SUBAPPLICATION AuxInput_Abscheider_UP (* Subapplication Type *)
  (* Standard: 61499-2 *)
  (* Version 1.0, 2023-02-06, franz *)
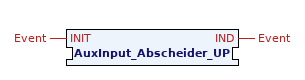
  EVENT_INPUT
    INIT;
  END_EVENT
  EVENT_OUTPUT
    IND;
  END_EVENT
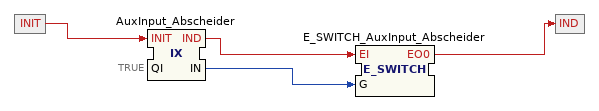
  FBS
    E_SWITCH_AuxInput_Abscheider : E_SWITCH;
    AuxInput_Abscheider : IX(QI := TRUE);
  END_FBS
  EVENT_CONNECTIONS
    AuxInput_Abscheider.IND TO E_SWITCH_AuxInput_Abscheider.EI;
    INIT TO AuxInput_Abscheider.INIT;
    E_SWITCH_AuxInput_Abscheider.EO0 TO IND;
  END_CONNECTIONS
  DATA_CONNECTIONS
    AuxInput_Abscheider.IN TO E_SWITCH_AuxInput_Abscheider.G;
  END_CONNECTIONS
END_SUBAPPLICATION
